INTERFACE I_Permissive EXTENDS I_Base

{attribute 'monitoring' := 'call'}
PROPERTY OK : BOOL
GET
END_GET
END_PROPERTY

METHOD Set
VAR_INPUT
	Index  : UDINT(0..9);
	Reason : STRING;
	Value  : BOOL;
END_VAR
END_METHOD

END_INTERFACE

(* stored: Version 1.1.0.1, ProductVersion 3.1.4026.18
   Itf I_Permissive: Id {daa32e67-53c9-4fc3-9c46-e7d7f3b46d9d}
   Property OK: Id {503d80e9-fff3-4a4c-8e11-2fa6322e7202}
   Get Get: Id {c3c6fcd1-aae0-4538-a6f9-b43248884bdd}
   Method Set: Id {f8659583-2db3-4caf-9c65-dd9d214495bb} *)
